Fanuc TP program (LS listing): PRT03_R01.LS

/PROG  PRT03_R01
/ATTR
OWNER		= MNEDITOR;
COMMENT		= "Main MH V4.0 335";
PROG_SIZE	= 2980;
CREATE		= DATE 18-11-21  TIME 05:37:40;
MODIFIED	= DATE 21-04-26  TIME 07:58:38;
FILE_NAME	= PRT01_R0;
VERSION		= 0;
LINE_COUNT	= 117;
MEMORY_SIZE	= 3448;
PROTECT		= READ_WRITE;
STORAGE		= SHADOW;
TCD:  STACK_SIZE	= 500,
      TASK_PRIORITY	= 50,
      TIME_SLICE	= 0,
      BUSY_LAMP_OFF	= 0,
      ABORT_REQUEST	= 0,
      PAUSE_REQUEST	= 0;
DEFAULT_GROUP	= 1,*,*,*,*;
CONTROL_CODE	= 00000000 00000000;
/APPL
  HANDLING : TRUE ;
/MN
   1:  !******************************** ;
   2:  !  GM METAL FORMING GLOBAL 4 S/W ;
   3:  !******************************** ;
   4:  !* Robot ID: IM010R01B01 ;
   5:  !*    F-196839 ;
   6:  !* Line: XXXXXXXX ;
   7:  !* Platform: XX ;
   8:  !* Tool ID: TOOL 03 ;
   9:  !* Part ID: PART 335 ;
  10:  !* Program: PRT03 ;
  11:  !* Application: MH PROCESS ;
  12:  !* SOURCE: TEMPLA12 ;
  13:  !******************************** ;
  14:  ! TEMPLA12: STANDARD PATH PROGRAM ;
  15:  ! TEMPLATE  FOR PICKING  FROM THE ;
  16:  ! EXIT  CONVEYOR  AND DROPING  ON ;
  17:  ! THE EOL CONVEYOR, WITH ONLY ONE ;
  18:  ! INTERFERENCE ZONE AT PICK. ;
  19:  !******************************** ;
  20:  ! 2016-02-14 GLOBAL-4 S/W REL 4.0 ;
  21:  !******************************** ;
  22:  !++++++++++++++++++++++++++++++++ ;
  23:  !INITIALIZE STYLE PROGRAM ;
  24:  !-------------------------------- ;
  25:   ;
  26:  TIMER[2]=RESET ;
  27:  TIMER[2]=START ;
  28:   ;
  29:  GO[1:0]=(3) ;
  30:  R[14]=100    ;
  31:  R[18]=.5    ;
  32:  R[19]=.5    ;
  33:  R[20]=1.5    ;
  34:   ;
  35:   ;
  36:  !INICIALIZE ALL TOOL DATA ;
  37:   ;
  38:  R[230]=1    ;
  39:  R[231]=1    ;
  40:  R[232]=1    ;
  41:  R[233]=0    ;
  42:  R[234]=0    ;
  43:  R[235]=0    ;
  44:  R[236]=1    ;
  45:   ;
  46:  ! R[142]=1 --> Vacuum Only ;
  47:  ! R[142]=2 --> Grippers Only ;
  48:  ! R[142]=3 --> Vacuum & Grippers ;
  49:   ;
  50:  R[142]=3    ;
  51:  R[211]=1    ;
  52:  R[212]=1    ;
  53:  R[213]=1    ;
  54:  R[214]=1    ;
  55:  !Check for correct Tool ;
  56:  CALL TL_CHK_KM(3) ;
  57:  !++++++++++++++++++++++++++++++++ ;
  58:   ;
  59:  !******************************** ;
  60:  !BEGINNING OF STYLE PROGRAM PATH ;
  61:  !******************************** ;
  62:  ! ;
  63:  !Move to Pick Pounce Core Moving ;
  64:  CALL PRT03POUNCE    ;
  65:   ;
  66:  !-------------------------------- ;
  67:  LBL[10:TOP OF LOOP] ;
  68:  REQUEST CONTINUE    ;
  69:   ;
  70:  ! Move to Home or Continue Cycle ;
  71:  SELECT R[150]=0,JMP LBL[20] ;
  72:         =15,JMP LBL[90] ;
  73:         ELSE,JMP LBL[10] ;
  74:   ;
  75:  !-------------------------------- ;
  76:  LBL[20:MOVE TO PICK] ;
  77:  ! Move to Pick ;
  78:  CALL PRT03PICK    ;
  79:   ;
  80:  !-------------------------------- ;
  81:  LBL[29:Pick Loop] ;
  82:  REQUEST CONTINUE    ;
  83:   ;
  84:  ! Move to PROC1, PROC2, or DROP2 ;
  85:  SELECT R[150]=15,JMP LBL[90] ;
  86:   ;
  87:  SELECT R[150]=0,JMP LBL[30] ;
  88:         =1,JMP LBL[50] ;
  89:         =3,JMP LBL[60] ;
  90:         ELSE,JMP LBL[29] ;
  91:  !-------------------------------- ;
  92:  LBL[30:Process1] ;
  93:  !Move to De-gate (Knife) Part ;
  94:  CALL PRT03PROC1    ;
  95:   ;
  96:  !-------------------------------- ;
  97:  LBL[39:Process1 Loop] ;
  98:  REQUEST CONTINUE    ;
  99:   ;
 100:  ! Move to PROC2, DROP1 or DROP2 ;
 101:  SELECT R[150]=2,JMP LBL[50] ;
 102:         =3,JMP LBL[60] ;
 103:         ELSE,JMP LBL[39] ;
 104:   ;
 105:  LBL[50:Drop1] ;
 106:  !Move to Drop Conveyor ;
 107:  CALL PRT03DROP1    ;
 108:  JMP LBL[90] ;
 109:   ;
 110:  LBL[60:Drop2] ;
 111:  !Move to Drop IM010R02 ;
 112:  CALL PRT03DROP2    ;
 113:  JMP LBL[90] ;
 114:   ;
 115:  LBL[90:END CYCLE] ;
 116:  !Move Home ;
 117:  MOVE TO HOME    ;
/POS
/END
